{attribute 'linkalways'} 
{attribute 'no_explicit_call' := 'This FB is a CLASS and must be accessed using methods or properties'}
{attribute 'enable_dynamic_creation'}
FUNCTION_BLOCK Node_RGBA_YELLOW EXTENDS VisionNode
VAR
    out : _TcVnVector4_LREAL;
END_VAR

METHOD PUBLIC  Clone : I_Node
VAR
	pNode : POINTER TO Node_RGBA_YELLOW;
END_VAR
pNode := __NEW(Node_RGBA_YELLOW);
Clone := pNode^;
END_METHOD

METHOD FB_init : BOOL
VAR_INPUT
	bInitRetains : BOOL; // if TRUE, the retain variables are initialized (warm start / cold start)
	bInCopyCode : BOOL;  // if TRUE, the instance afterwards gets moved into the copy code (online change)
END_VAR
AddOutput('out', out);
END_METHOD

METHOD PROTECTED OnExecute : HRESULT
out.Value := GVL_COLOURS.RGBA_YELLOW;
END_METHOD

METHOD PUBLIC PreExecutionCheck
VAR_INPUT
	Check : I_PreExecutionChecks;
END_VAR
END_METHOD

END_FUNCTION_BLOCK

(* stored: Version 1.1.0.1, ProductVersion 3.1.4024.13
   POU Node_RGBA_YELLOW: Id {8dcf2775-1f76-0f1f-3d47-dc3df9478b88}, SpecialFunc None
   Folder Constructor: Id {83527210-c9a6-0c5b-177a-8b23486ac17c}
   Method Clone: Id {703f1653-9754-097c-1d13-49cecc0aaabb}
   Method FB_init: Id {3b8dca83-7d84-050a-289a-ff825e30dece}
   Method OnExecute: Id {7c4dc1a6-eb57-0a19-3737-49e551b1f47a}
   Method PreExecutionCheck: Id {133ba043-d598-0f44-1e20-f6f99943fc2d} *)
